// Mitsubishi GX Works2 project: ventilation_v01   PLC: FX3G
// Базовая структура управления вентиляциооной установкой

// global labels: Global1
VAR_GLOBAL
  xStart AT M15 : BOOL;  (* Переменная разрешения на работу установки *)
  xSeason AT M16 : BOOL;  (* Определение сезона 0 - Зима 1 - Лето *)
  xAlarm AT M1 : BOOL;  (* Общий статус Аварий 0 - нет 1 - Авария *)
  xWarning AT M2 : BOOL;  (* Общий статус предупреждений 0 - нет 1 - есть предупреждения *)
  dI_AlFreeze AT X000 : BOOL;  (* Авария термостата заморозки *)
  xAlarmSensors AT M7 : BOOL;  (* Общая аврия Датчиков - всне диапазона *)
  dI_AlPumpWater AT X001 : BOOL;  (* Авария насоса (сработка защиты) *)
  dI_AlMotorSupply AT X002 : BOOL;  (* Авария реле Вентилятора Притока *)
  dI_AlMotorExhaust AT X003 : BOOL;  (* Авария реле Вентилятора Вытяжки *)
  dI_WarnPresFilterSupply AT X007 : BOOL;  (* Авария пресостата фильтра Притока *)
  dI_WarnPresFilterExaust AT X006 : BOOL;  (* Авария пресостата фильтра Вытяжки *)
  dI_AlPresMotorSupply AT X004 : BOOL;  (* Авария пресостата вентилятора Притока *)
  dI_AlPresMotorExhaust AT X005 : BOOL;  (* Авария пресостата вентилятора Вытяжки *)
  xAlarmWarmWater AT M8 : BOOL;  (* Авария снижения температуры теплоносителя темплообменника - Требуется прогрев *)
  wDeltaTempOut AT D11 : INT;  (* Значение смещения показаний датчика (корректировка) *)
  wDeltaTempInRoom AT D10 : INT;  (* Значение смещения показаний датчика (корректировка) *)
  wDeltaTempFromRoom AT D9 : INT;  (* Значение смещения показаний датчика (корректировка) *)
  wDeltaTempEmpty AT D8 : INT;  (* Значение смещения показаний датчика (корректировка) *)
  xAlarmSensorOut AT M6 : BOOL;  (* Авария датчика Наружней температуры *)
  xAlarmSensorSupply AT M5 : BOOL;  (* Авария датчика температуры Подачи В помещение *)
  xAlarmSensorRecup AT M4 : BOOL;  (* Авария датчика температуры забираемого ИЗ помещения *)
  iR_TempOut AT D6 : WORD;  (* Значение сопротивление линии связи резистивного датчика *)
  iR_TempInRoom AT D5 : WORD;  (* Значение сопротивление линии связи резистивного датчика *)
  iR_TempFromRoom AT D4 : WORD;  (* Значение сопротивление линии связи резистивного датчика *)
  iRTempEmpty AT D7 : WORD;  (* Значение сопротивление линии связи резистивного датчика *)
  dO_PumpStart AT Y004 : BOOL;  (* Разрешение на работу Насоса контура водяного теплообменника *)
  dO_SupplyMotorStart AT Y003 : BOOL;  (* Разрешение на запуск Вентилятора Притока *)
  dO_ExhaustMotorStart AT Y001 : BOOL;  (* Разрешение на запуск Вентилятора Вытяжки *)
  dO_SupplyDamperStart AT Y002 : BOOL;  (* Разрешение на открытие Заслонки Притока *)
  dO_ExhaustDamperStart AT Y000 : BOOL;  (* Разрешение на открытие Заслонки Вытяжки *)
  iEmpty2 AT D3 : INT;  (* Значение задержки пуска Вентилятора Притока *)
  iEmpty AT D1 : INT;  (* Значение задержки пуска Вентилятора Вытяжки *)
  xUserStart AT M21 : BOOL;  (* Переменная изменяемая Пользователем для разрешения работы *)
  xUserSeason AT M22 : BOOL;  (* Переменная изменяемая Пользователем для выбора Сезона *)
  xUserArarmReset AT M23 : BOOL;  (* Переменная изменяемая Пользователем для сброса общего флага Аварий *)
  xAlarmCritical AT M0 : BOOL;  (* Cтатус критических Аварий 0 - нет 1 - Авария *)
  xInit AT M31 : BOOL;  (* Переменная разрешающая иницилизацию при старте *)
  aI_TempOut AT D14 : INT;  (* AI_0 Датчик наружней температуры D8033 *)
  aI_TempSupply AT D15 : INT;  (* AI_1 Датчик притока (температуры подачи в помещение)  D8031 *)
  aI_TempWater AT D16 : INT;  (* AI_2 Датчик обратной воды  D8032 *)
  aI_TempRecupOut AT D17 : INT;  (* AI_3 Датчик температуры за рекуператором  D8030 *)
  aO_1 AT D8050 : REAL;  (* AO_ Первый аналоговый D8050 *)
  aO_2 AT D8051 : REAL;  (* AO_ Второй аналоговый выход D8051 *)
  iUserTempSummer AT D128 : INT;  (* Температура перехода на летний режим *)
  iUserTemWinter AT D129 : INT;  (* Температура перехода на зимний режим *)
  aI_TempFromRoom AT D18 : INT;  (* AI_4 Датчик вытяжной температуры из помещения D8034 *)
  iUserAccess AT D40 : WORD;  (* Уровень доступа текущего пользователя *)
  iUserSetTSupply AT D130 : INT;  (* Уставка заданная пользователем *)
  testTempOut AT D41 : REAL;  (* Тестирование перехода   Зима/Лето *)
  iSetpointTempSupply AT R550 : INT;  (* Уставка температуры подачи Системная *)
  iUserSetTWater AT D131 : INT;  (* Уставка контроля температуры теплоносителя (вода) *)
  iUserSetTGlycol AT D132 : INT;  (* Уставка контроля температуры теплоносителя гликоль *)
  iUserSetTAlarmWaterStop AT D133 : INT;  (* Уставка контроля температуры Аварии *)
  xArarmReset AT M30 : BOOL;  (* Переменная сбрасывающая все Аварии *)
  xUserStartBut AT M20 : BOOL;
  xAlarmFreeze AT M3 : BOOL;
  TOF_ten : TOF_10;
  TON_ten : TON_10;  (* Таймер с задержкой включения Если управляющий сигнал становиться 0 - таймер прерывается *)
  wUserDelayExause AT D140 : WORD;  (* Время задержки для запуска Вытяжного вентилятора *)
  wUserDelayDamper AT D142 : WORD;  (* Время задержки для открытия заслонки *)
  wUserDelaySupply AT D141 : WORD;  (* Время задержки для запуска Приточного вентилятора *)
  wUserTimeWarmUp AT D143 : WORD;  (* Время прогрева перед стартом и при сработке Аварии по Т теплоностителя *)
  xHeatBeforeStart AT M33 : BOOL;  (* Прогрев перед стартом 0 - не нужен 1 - Требуется *)
  TP_ten : TP_10;  (* Создается импульс заданной продолжительности *)
  xPIDModeAir AT M51 : BOOL;  (* Определяет режим работы PID регулятора поддержания Т приточного воздуха 1 - auto 0 - manual (по установленным пользователем параметрам) *)
  xPIDModeWater AT M52 : BOOL;  (* Определяет режим работы PID регулятора поддержания Т обратной воды 1 - auto 0 - manual (по установленным пользователем параметрам) *)
  xPIDStatus AT M50 : BOOL;  (* Режим работы PID регулятора: 0 - контроль Т обратной воды 1- контроль Т притока *)
  iPIDAir_out AT D42 : INT;  (* результат работы PID регулятора поддержания Т воздуха в приточном канале *)
  iPIDWater_out AT D43 : INT;  (* результат работы PID регулятора поддержания T воды (обратной) *)
  xPIDAirTypeAuto AT M53 : BOOL;  (* Определяет тип автоматической работы по Воздуху 1 - циклами  0 - шагами *)
  xPIDWTypeAuto AT M54 : BOOL;  (* Определяет тип автоматической работы по Воде 1 - циклами  0 - шагами *)
  wPIDAirKp AT D150 : WORD;  (* Пропорциональный коэфициент - PID Air *)
  wPIDAirTi AT D151 : WORD;  (* Время Интегрирования - PID Air *)
  wPIDAirKd AT D152 : WORD;  (* Диференциальный коэфициент - PID Air *)
  wPIDAirTd AT D153 : WORD;  (* Время Диференцирования - PID Air *)
  wPIDWaterKp AT D155 : WORD;  (* Пропорциональный коэфициент - PID Water *)
  wPIDWaterTi AT D156 : WORD;  (* Время Интегрирования - PID Water *)
  wPIDWaterKd AT D157 : WORD;  (* Диференциальный коэфициент - PID Water *)
  wPIDWaterTd AT D158 : WORD;  (* Время Диференцирования - PID Water *)
  wPIDAirDeltaAtune AT D154 : WORD;  (* Величина отклонения от Уставки при автонастройке (зона нечувствительности) - PID Air *)
  wPIDWDeltaAtune AT D159 : WORD;  (* Величина отклонения от Уставки при автонастройке (зона нечувствительности)  - PID Water *)
END_VAR

// task Task_01 (event TRUE, interval 0, priority 31): POU_01
// task Init (event M8002, interval 0, priority 24): Init
// task Process (event FALSE, interval T#150ms, priority 29): Process
// user libraries (not included): alarmManager, tempControl

PROGRAM Init
VAR
  inputType : BOOL;
  aInit : A_init;
END_VAR
(* PID Air Supply *)
R500 := 1000; (* Sampling Time - время обработки *)
R501 := 2#0000_0000_0000_0001; (* Первый  бит определят тип регулировки - 1 нагрев 0 - охлаждение *)
IF xPIDModeAir THEN 
	(* R501 := SRB( R501 , 4 , TRUE ); *)
	(* R501 := SRB( R501 , 5 , TRUE ); *)
	(* IF xPIDAirTypeAuto THEN R501 := SRB( R501 , 6 , TRUE );  END_IF; *)
	;
END_IF;

R502 := 30; (* Входной фильтр *)
(*R503 - Kp Пропорциональный коэфициент  *)
(*R504 - Ti Время Интегрирования ms *)
(*R505 - Kd Диференциальный коэфициент   *)
(*R506 - Td Время диференцирования ms  *)
(*R507 - R520 Используется PID регулятором для внутренних расчетов *)
R522 := 1000; (*Верхний выходной предел  *)
R523 := 0; (*Нижний выходной предел  *)
(* Настройки для авторегулировки  *)
R525 :=  1; (* Зона нечуствительности при автонастройке - отклонение от Уставки *)
R526 := R522; (*Верхний выходной предел  *)
R527 := 0; (*Нижний выходной предел  *) 

(* PID Water return *)
R600 := 1000; (* Sampling Time - время обработки *)
R601 := 2#0000_0000_0000_0001;
IF xPIDModeWater THEN 
	R601 := 2#0000_0000_0011_0001;
	IF xPIDWTypeAuto THEN R601 := 2#0000_0000_0111_0001; END_IF;
END_IF;
R602 := 30; (* Входной фильтр *)
(*R503 - Kp Пропорциональный коэфициент  *)
(*R504 - Ti Время Интегрирования ms *)
(*R505 - Kd Диференциальный коэфициент   *)
(*R506 - Td Время диференцирования ms  *)
(*R507 - R520 Используется PID регулятором для внутренних расчетов *)
R622 := 1000; (*Верхний выходной предел  *)
R623 := 0; (*Нижний выходной предел  *)
(* Настройки для авторегулировки  *)
R625 :=  1; (* Зона нечуствительности при автонастройке - отклонение от Уставки *)
R626 := R522; (*Верхний выходной предел  *)
R627 := 0; (*Нижний выходной предел  *) 

(* Critical Alarm signals*)
	aInit(iNum:= 0 ,iSeverity:= 3 ,iProcess:= 1 ,xLatch:= TRUE ,xBuzzer:= TRUE , xLock:= TRUE ); (* Freeze *)
	aInit(iNum:= 1 ,iSeverity:= 3 ,iProcess:= 1 ,xLatch:= TRUE ,xBuzzer:= TRUE , xLock:= TRUE ); (* Fire *)
	aInit(iNum:= 2 ,iSeverity:= 3 ,iProcess:= 3 ,xLatch:= FALSE ,xBuzzer:= TRUE , xLock:= TRUE ); (* Wurming Up *)
	aInit(iNum:= 3 ,iSeverity:= 3 ,iProcess:= 3 ,xLatch:= FALSE ,xBuzzer:= TRUE , xLock:= TRUE ); (* Alarm pump*)
	aInit(iNum:= 4 ,iSeverity:= 3 ,iProcess:= 4 ,xLatch:= FALSE ,xBuzzer:= TRUE , xLock:= TRUE ); (* Alarm Frequency Steam Generation *)
	aInit(iNum:= 5 ,iSeverity:= 3 ,iProcess:= 4 ,xLatch:= FALSE ,xBuzzer:= TRUE , xLock:= TRUE ); (* Alarm Motor Supply *)
	aInit(iNum:= 6 ,iSeverity:= 3 ,iProcess:= 4 ,xLatch:= FALSE ,xBuzzer:= TRUE , xLock:= TRUE ); (* Alarm Motor Exhaust*)
	aInit(iNum:= 7 ,iSeverity:= 3 ,iProcess:= 4 ,xLatch:= FALSE ,xBuzzer:= TRUE , xLock:= TRUE ); (* Alarm Motor Supply Presure*)
	aInit(iNum:= 8 ,iSeverity:= 3 ,iProcess:= 4 ,xLatch:= FALSE ,xBuzzer:= TRUE , xLock:= TRUE ); (* Alarm Motor Exhaust Presure*)
	
(*Temperature Sersors connect*)
aInit(iNum:= 9, iSeverity:= 2 ,iProcess:= 2 ,xLatch:= FALSE ,xBuzzer:= FALSE, xLock:= TRUE ); (* Common sensors Alarm  *)
aInit(iNum:= 10, iSeverity:= 2 ,iProcess:= 2 ,xLatch:= FALSE ,xBuzzer:= FALSE, xLock:= TRUE ); (* D8031 - AI02 Temp Supply Room  *)
aInit(iNum:= 11, iSeverity:= 2 ,iProcess:= 2 ,xLatch:= FALSE ,xBuzzer:= FALSE , xLock:= TRUE ); (* D8030 - AI01 Temp Out *)
aInit(iNum:= 12, iSeverity:= 2 ,iProcess:= 2 ,xLatch:= FALSE ,xBuzzer:= FALSE , xLock:= TRUE ); (* D8031 - AI03 Temp Water Return *)
aInit(iNum:= 13, iSeverity:= 2 ,iProcess:= 2 ,xLatch:= FALSE ,xBuzzer:= FALSE , xLock:= TRUE ); (* D8033 - AI04 Temp After Recup  *)

(*Presure Sensors*)
aInit(iNum:= 14, iSeverity:= 1 ,iProcess:= 5 ,xLatch:= FALSE ,xBuzzer:= FALSE , xLock:= FALSE ); (* Supply Presure Warning *)
aInit(iNum:= 15, iSeverity:= 1 ,iProcess:= 5 ,xLatch:= FALSE ,xBuzzer:= FALSE , xLock:= FALSE ); (* Exhaust Presure Warning *)
END_PROGRAM

PROGRAM POU_01
VAR
  iStep : INT;
  localSeasonTriger : BOOL;
  icountMin : INT;
  init : INT;
  currentTemp : INT;
  couner : INT;
  aReset : A_reset;
  aStatus : A_status;
  TON_Exhaust : TON_10;
  TON_Suply : TON_10;
  TON_Dumper : TON_10;
  timeDelayExause : TIME;
  timeDelaySupply : TIME;
  timeDelayDamper : TIME;
  plWarmUp : BOOL;  (* импульс на прогрев *)
  timeDelayWarming : TIME;
  plDump : BOOL;  (* импульс открытия закрытия заслонки *)
END_VAR
 (* RST( MEP( xManualWorks ) , xAutoWorks );
RST( MEP(xAutoWorks ) ,xManualWorks  );  *)
(* System can work only in one state Auto or Manual There is constol change*)

(*	RST( MEF(xStart)  , TON_Dumper ); *)  (* Сброс таймера ожидания задержки открытия заслонки  *)

 		IF xInit = 0 OR xAlarm =1 THEN  iStep := 0 ; (* Проверяем была ли выполнена инициализация xInit = 1 Ули была то переходим на шаг 10 если нет - на шаг 0 *)
 		ELSE 
 			IF xStart  AND xHeatBeforeStart  THEN iStep := 20; ELSE iStep := 10; END_IF; (* Проверяем нужнен ли прогрев перед стартом если да то шаг 20 иначе шаг 10  *)
 		END_IF; 

CASE iStep OF
	0: (* Init  - Инициализация Задаем начальные значения переменным*)
		dO_ExhaustDamperStart := 0;
		dO_SupplyDamperStart := 0;
		dO_ExhaustMotorStart := 0;
		dO_SupplyMotorStart := 0;
		
		timeDelayDamper := (WORD_TO_TIME(wUserDelayDamper) * 1000);
		timeDelayExause := (WORD_TO_TIME(wUserDelayExause) * 1000);
		timeDelaySupply := (WORD_TO_TIME(wUserDelaySupply) * 1000);
		timeDelayWarming := (WORD_TO_TIME(wUserTimeWarmUp) * 1000);
		
		IF NOT xAlarmWarmWater THEN 
			aO_1 := 0.0;
			aO_2 := 0.0;
		END_IF;
		xInit := 1;
		iStep := 10;

	
	10: (* Base  Manage *)
	(* После появления сигнала xStart происходит полеледовательный пуск установки с заданными задержками*)
	TON_Dumper(IN:= xStart , PT:=  timeDelayDamper  ,Q:= dO_ExhaustDamperStart ); 
	(* IF MEP(plDump ) THEN  dO_ExhaustDamperStart :=1; END_IF; *)
	(* IF MEF(plDump ) THEN  dO_ExhaustDamperStart :=0; END_IF; *)
		
	TON_Exhaust(IN:= dO_ExhaustDamperStart, PT:= timeDelayExause ,Q:= dO_ExhaustMotorStart ); 
	dO_SupplyDamperStart := dO_ExhaustMotorStart ;
	TON_Suply(IN:= dO_SupplyDamperStart , PT:= timeDelayDamper ,Q:= dO_SupplyMotorStart);
	
			
	(* Поддержание температуры воздуха в приточном канале *)
	PID( (xStart AND xSeason) , iSetpointTempSupply , aI_TempSupply,  R500 , iPIDAir_out);
	
		(* Поддержание температуры воды (обраной) при ожидании пуска*)
	PID(
	 (NOT xStart AND xSeason AND dO_SupplyDamperStart ) , (* Разрешение на работу *)
	iUserSetTWater, (* Уставка *)
	aI_TempWater ,  (* Текущее значение *)
	R600 , (* Первая ячейка о бласти памяти для определения настроек регулятора*)
	iPIDWater_out (* Сохранение результата *)
	);
	
	IF xSeason THEN
			IF xStart THEN
				aO_1 := INT_TO_REAL( iPIDAir_out );
				ELSE 
				aO_1 := INT_TO_REAL( iPIDWater_out);
			END_IF;
		ELSE 
		aO_1 := 0.0;
	END_IF;
	
	20: (* Warming Up befor Start *)
	aO_1 :=   warmCalc( INT_TO_REAL (aI_TempOut),  INT_TO_REAL (aI_TempWater), 100.0, 5.0 ); (* Вычисляем % открытия клапана при прогреве по Т улицы и Т теплоносителя *)
	TP_ten(IN:= xHeatBeforeStart , PT:= timeDelayWarming , Q:= plWarmUp );
	IF MEF(plWarmUp ) THEN 
		xHeatBeforeStart := 0; 
		aO_1 := (warmCalc( INT_TO_REAL (aI_TempOut),  INT_TO_REAL (aI_TempWater), 80.0, 30.0 ) / 2.0 );
	END_IF;
	
	
	
	100: (* Alarm *)
		;
	END_CASE;



(*	
D500 := D100Z1;

IF MEP( M8013) AND xUserStart = TRUE  THEN
	icountMin := icountMin +1;
	IF icountMin =8 THEN
		icountMin := 0;

	END_IF;
END_IF; 
*)
END_PROGRAM

PROGRAM Process
VAR
  aInit : A_init;
  aSet : A_set;
  TP_RST : TP;
  start_RST : BOOL;
  start_Warm : BOOL;
  aStatus : A_status;
  aRST : A_reset;
END_VAR
(*All proccess that works constantly - monit alarms, statuses and so on *)
(* Выполняем регистрацию события объявленного в программе Init при выполнении определенного (указываем при вызове) условия *)

(* Input  sensors Error - not data or conection from sensors conection*)
 (*iNum - number registred in Init programm Alarm  xState - condition for execution*)
 aSet(iNum:= 9, xState:=  ((D8030 = 4984) OR (D8031 = 4984) OR (D8032 = 4984) OR (D8033 = 4984) ), Q:= xAlarmSensors);
 aSet(iNum:= 10, xState:=  (D8033 = 4984), Q:= xAlarmSensorOut );
 aSet(iNum:= 11, xState:=  (D8031 = 4984), Q:= xAlarmSensorSupply );
 aSet(iNum:= 13, xState:=  (D8030 = 4984), Q:= xAlarmSensorRecup );

	IF NOT (D8033 = 4984) THEN aI_TempOut := LIMITATION(-500, D8033, 500);  ELSE aI_TempOut := 990; END_IF ;   (*Проверяем входной порт D8030 на ошибку и сохраняем значение входа в 
	переменную aI_TempOut Если ошибка есть назначаем - 999*)
	IF NOT (D8031 = 4984) THEN aI_TempSupply := (D8031 + 1000); ELSE aI_TempSupply := 999; END_IF ;    (*aI_TempSupply *)
	IF NOT (D8032 = 4984) THEN aI_TempWater := (D8032 + D8031 +500 ); ELSE aI_TempWater := 999; END_IF ;   (*aI_TempWater *)
	IF NOT (D8030 = 4984) THEN aI_TempRecupOut:= D8030; ELSE aI_TempRecupOut:= 999; END_IF ;   (*aI_TempFromRoom *)	

 (*reset ALL Alarms *)
 TP_RST(IN:=xUserArarmReset , PT:= T#500ms ,Q:= xArarmReset );
 aRST(reset:= xArarmReset );
IF xArarmReset THEN xUserArarmReset := 0; END_IF;

 (*registration Alarms from Digital Input*)
 aSet(iNum:= 0, xState:=  (NOT X000), Q:= xAlarmFreeze);
 aSet(iNum:= 2, xState:=  ((aI_TempWater <( iUserSetTAlarmWaterStop * 10)) OR xAlarmFreeze), Q:= xAlarmWarmWater);
 
 
  aStatus(ALARM:= xAlarm ,CRITICAL:=xAlarmCritical );
 IF MEP(xAlarmCritical) THEN xUserStart := 0; END_IF;
 	
(*Control of changes in the Season variable depending on the Outdoor Temperature *)
xSeason := SeasonControl( aI_TempOut , (iUserTemWinter * 10) , (iUserTempSummer * 10),  xUserSeason );
		IF MEP(xSeason) OR MEF(xSeason) THEN
			xUserSeason :=  xSeason ;
			IF MEP(xSeason) THEN dO_PumpStart := 1; END_IF;
			IF MEF(xSeason) THEN dO_PumpStart := 0; END_IF;
				IF xSeason THEN 
					;
				END_IF;
(*
				IF xSeason =1 THEN
						dO_PumpStart := 1;
					ELSE 
						dO_PumpStart := 0;
				END_IF; 
*)
			END_IF;
			
(* Control PID Settings *)
IF MEP(xStart) THEN (* Проверка настроек PID регулятора в момент включения *)
	iSetpointTempSupply := iUserSetTSupply * 10;
	R501 := 2#0000_0000_0111_0001;
	
	(* R501 := SRB( R501 , 4 , TRUE ); *)
	(* R501 := SRB( R501 , 5 , TRUE ); *)
	(* IF xPIDAirTypeAuto THEN R501 := SRB( R501 , 6 , TRUE );  END_IF; *)
		R503 := wPIDAirKp;
		R504 := wPIDAirTi;
		R505 := wPIDAirKd;
		R506 := wPIDAirTd;
		R525 := wPIDAirDeltaAtune;
	END_IF;
	
	IF MEF(xStart) AND (NOT xPIDStatus)THEN (* Проверка настроек PID регулятора в момент включения *)
	R601 := SRB( R601 , 4 , TRUE );  
	R601 := SRB( R601 , 5 , TRUE ); 
	IF xPIDWTypeAuto THEN R601 := SRB( R601 , 6 , TRUE );  END_IF;
		R603 := wPIDWaterKp;
		R604 := wPIDWaterTi;
		R605 := wPIDWaterKd;
		R606 := wPIDWaterTd;
		R625 := wPIDWDeltaAtune;
	END_IF;
	

(*Start / Stop Control *)
TP_RST(IN:= MEF(xUserStartBut) , PT:= T#1s, Q:= start_RST); (* Detect rare impuls button and set start_RST =1 on 1 sec *)
IF start_RST = 1 AND xUserStart = 1 THEN xUserStart := 0; END_IF; (* reset xUserStart valuable *)
IF (xUserStart OR xUserStartBut) AND (NOT xAlarmCritical) THEN xStart := 1; ELSE xStart :=0; END_IF;
IF MEP(xStart) AND xSeason THEN xHeatBeforeStart := 1; END_IF;
	
		
(*Freeze Alarm *)

(* TP_RST(IN:= MEP(xAlarmWarmWater) , PT:= T#15s, Q:= start_Warm); *)
(* Принудительно удерживаем клапан управления теплоносителем в открытом состоянии *)
TOF_ten(IN:= xAlarmWarmWater , PT:= T#6s ,Q:= start_Warm );
	IF start_Warm THEN 
		MOV(start_Warm , 100,  D8050 );
	ELSE 
		MOV((NOT start_Warm) , 0,  D8050 );
	END_IF; 

(* fbAmSet(iNum:= 0, xState:= (NOT X000) ); *)


(* PLS( xUserArarmReset , xArarmReset); *)
(* IF xArarmReset THEN fbAmRST( ); END_IF; *)
(* *)

(* *)

(* *)
;
(* *)
END_PROGRAM

FUNCTION SeasonControl
VAR_INPUT
  tempOut : INT;  (* Temp Outdore - Температура наружнего воздуха *)
  tempWinter : INT;  (* Temp for switch on Winter - Уставка перехода на Зимний режим *)
  tempSummer : INT;  (* Temp for switch on Summer - Уставка перехода на летний режим *)
  triger : BOOL;  (* 1 - was switch to winter 0 - was switch to summer *)
END_VAR
IF tempOut  <  tempWinter THEN 
		SeasonControl := 1; (* Output  Set flag - 1  to force switching to Winter *)
	ELSE 
		IF tempOut  > tempSummer THEN 
			SeasonControl := 0; (* Output  Set flag - 0  to force switching to Summer*)
		ELSE 
			SeasonControl := triger; (* Don't change r*)
		END_IF;

	END_IF;
END_FUNCTION

FUNCTION TestFunction
TestFunction := TRUE;
END_FUNCTION
